PROGRAM Notes
VAR
END_VAR

// Write notes here

// Comment out

END_PROGRAM

(* stored: Version 1.1.0.1, ProductVersion 3.1.4024.13
   POU Notes: Id {65549388-3fcb-437a-a9ec-b8ef626c5b06}, SpecialFunc None *)
